// TwinCAT 3 PLC project Library
// Title: Tc3_Logging
// Company: www.peterzerlauth.com
// Author: Peter Zerlauth
// ProjectVersion: 0.0.0.0
// ProgramVersion: 3.1.4026.19
// libraries:
//   Tc2_Standard, * (Beckhoff Automation GmbH)
//   Tc2_System, * (Beckhoff Automation GmbH)
//   Tc2_Utilities, * (Beckhoff Automation GmbH)
//   Tc3_EventLogger, * (Beckhoff Automation GmbH)
//   Tc3_Module, * (Beckhoff Automation GmbH)
// project tree:
//   Helpers/ F_Format.TcPOU, F_InstancePath.TcPOU (not stored)
//   Logger/ FB_Argument.TcPOU, FB_Logger.TcPOU, I_Argument.TcIO
//   Logging/ E_LogLevel.TcDUT (not stored), FB_Logging.TcPOU, I_Logger.TcIO, I_Logging.TcIO, ST_Message.TcDUT (not stored)
//   Project Information/ F_GetCompany.TcPOU (not stored), F_GetTitle.TcPOU (not stored), F_GetVersion.TcPOU
//   TcLogging/ FB_TcLogging.TcPOU
//   Version/ Global_Version.TcGVL
// (motion and I/O tree: see PLC project plc01)
// real-time tasks:
//   TASK SlowTask: cycle T#20ms, priority 20, ADS port 350
//   TASK FastTask: cycle T#1ms, priority 1, ADS port 351

// ---- Version/Global_Version.TcGVL
{attribute 'TcGenerated'}
{attribute 'no-analysis'}
{attribute 'linkalways'}
// This function has been automatically generated from the project information.
VAR_GLOBAL CONSTANT
	{attribute 'const_non_replaced'}
	stLibVersion_Tc3_Logging : ST_LibVersion := (iMajor := 0, iMinor := 0, iBuild := 0, iRevision := 0, nFlags := 0, sVersion := '0.0.0.0');
END_VAR

// ---- Logger/I_Argument.TcIO
INTERFACE I_Argument

METHOD PUBLIC M_AddBOOL : I_Argument
VAR_INPUT
	nValue:				LINT;
END_VAR
END_METHOD

METHOD PUBLIC M_AddINT : I_Argument
VAR_INPUT
	nValue:				LINT;
END_VAR
END_METHOD

METHOD PUBLIC M_AddREAL : I_Argument
VAR_INPUT
	fValue:				LREAL;
	nDecimals:			USINT;
END_VAR
END_METHOD

METHOD PUBLIC M_AddSTRING : I_Argument
VAR_INPUT
	sValue:				STRING(255);
END_VAR
END_METHOD

METHOD PUBLIC M_AddTIME : I_Argument
VAR_INPUT
	tValue:				TIME;
END_VAR
END_METHOD

METHOD PUBLIC M_Clear : I_Argument
VAR_INPUT
END_VAR
END_METHOD

PROPERTY PUBLIC P_Value : string(255)
GET
END_GET
END_PROPERTY

END_INTERFACE

// ---- Logging/I_Logger.TcIO
INTERFACE I_Logger

METHOD PUBLIC M_AddBOOL
VAR_INPUT
	nValue:				LINT;
END_VAR
END_METHOD

METHOD PUBLIC M_AddINT
VAR_INPUT
	nValue:				LINT;
END_VAR
END_METHOD

METHOD PUBLIC M_AddREAL
VAR_INPUT
	fValue:				LREAL;
	nDecimals:			USINT;
END_VAR
END_METHOD

METHOD PUBLIC M_AddSTRING
VAR_INPUT
	sValue:				STRING(255);
END_VAR
END_METHOD

METHOD PUBLIC M_AddTIME
VAR_INPUT
	tValue:				TIME;
END_VAR
END_METHOD

METHOD PUBLIC M_Debug : BOOL
VAR_INPUT
	sMessage:			STRING(255);
END_VAR
END_METHOD

METHOD PUBLIC M_Error : BOOL
VAR_INPUT
	nID:				UDINT;
	sMessage:			STRING(255);
END_VAR
END_METHOD

METHOD PUBLIC M_Fatal : BOOL
VAR_INPUT
	nID:				UDINT;
	sMessage:			STRING(255);
END_VAR
END_METHOD

METHOD PUBLIC M_Info : BOOL
VAR_INPUT
	nID:				UDINT;
	sMessage:			STRING(255);
END_VAR
END_METHOD

METHOD PUBLIC M_Warn : BOOL
VAR_INPUT
	nID:				UDINT;
	sMessage:			STRING(255);
END_VAR
END_METHOD

END_INTERFACE

// ---- Logging/I_Logging.TcIO
INTERFACE I_Logging

METHOD PUBLIC M_Attach : BOOL
VAR_INPUT
	iLogging:				I_Logging;
END_VAR
END_METHOD

METHOD PUBLIC M_Log : BOOL
VAR_INPUT
	stMessage:			ST_Message;
END_VAR
END_METHOD

PROPERTY PUBLIC P_LogLevel : E_LogLevel
GET
END_GET
SET
END_SET
END_PROPERTY

END_INTERFACE

// ---- Helpers/F_Format.TcPOU
FUNCTION F_Format : STRING(255)
VAR_INPUT
    sMessage:				STRING(255);
    sArguments:				STRING(255);	// Arguments are separated by $R 
END_VAR
VAR
    sArg:					STRING; 	// single argument
    nPosition:				INT;         	// Position of the $R delimiter
    nPlaceholder:			INT;         	// Position of the %s placeholder
END_VAR

// replace placeholders with arguments
F_Format := sMessage;

IF sArguments = '' THEN
    RETURN;
END_IF

nPosition := FIND(sArguments, '$R');
WHILE nPosition > 0 DO
    
    sArg := LEFT(sArguments, nPosition - 1);
    
    nPlaceholder := FIND(F_Format, '%s');
    IF nPlaceholder > 0 THEN
        F_Format := REPLACE(F_Format, sArg, 2, nPlaceholder);
    ELSE
        RETURN;
    END_IF
	
    sArguments := DELETE(sArguments, nPosition, 1);
    nPosition := FIND(sArguments, '$R');
    
END_WHILE

END_FUNCTION

// ---- Logger/FB_Argument.TcPOU
FUNCTION_BLOCK FB_Argument IMPLEMENTS I_Argument
VAR_INPUT
END_VAR
VAR_OUTPUT
END_VAR
VAR
	sValue:					STRING(255); 
END_VAR

METHOD PUBLIC M_AddBOOL : I_Argument
VAR_INPUT
	nValue:				LINT;
END_VAR
sValue:= LINT_TO_STRING(nValue);			// convert
sValue:= CONCAT(sValue, '$R');				// add separator
sValue:= CONCAT(sValue, sValue);	// add new arg
M_AddBOOL:= THIS^;
END_METHOD

METHOD PUBLIC M_AddINT : I_Argument
VAR_INPUT
	nValue:				LINT;
END_VAR
VAR
	sTemp: 			STRING;
END_VAR
sTemp:= LINT_TO_STRING(nValue);			// convert
sTemp:= CONCAT(sTemp, '$R');				// add separator
sValue:= CONCAT(sValue, sTemp);	// add new arg
M_AddINT:= THIS^;
END_METHOD

METHOD PUBLIC M_AddREAL : I_Argument
VAR_INPUT
	fValue:				LREAL;
	nDecimals:			USINT;
END_VAR
VAR
	sTemp: 			STRING;
END_VAR
sTemp:= LREAL_TO_FMTSTR(fValue, nDecimals, TRUE);		// convert
sTemp:= CONCAT(sTemp, '$R');							// add separator
sValue:= CONCAT(sValue, sTemp);				// add new arg
M_AddREAL:= THIS^;
END_METHOD

METHOD PUBLIC M_AddSTRING : I_Argument
VAR_INPUT
	sValue:				STRING(255);
END_VAR
THIS^.sValue:= CONCAT(THIS^.sValue, CONCAT(sValue, '$R'));				// add separator 
M_AddSTRING:= THIS^;
END_METHOD

METHOD PUBLIC M_AddTIME : I_Argument
VAR_INPUT
	tValue:				TIME;
END_VAR
VAR
	sTemp: 			STRING;
END_VAR
sValue:= CONCAT(TIME_TO_STRING(tValue), '$R');				// add separator
sTemp:= CONCAT(sValue, sTemp);	// add new arg
M_AddTIME:= THIS^;
END_METHOD

METHOD PUBLIC M_Clear : I_Argument
VAR_INPUT
END_VAR
sValue:= '';
M_Clear:= THIS^;
END_METHOD

PROPERTY PUBLIC P_Value : string(255)
GET
P_Value:= sValue;
END_GET
END_PROPERTY

END_FUNCTION_BLOCK

// ---- Logger/FB_Logger.TcPOU
{attribute 'reflection'} 
FUNCTION_BLOCK FB_Logger
VAR_INPUT
	iLogging:			I_Logging;
END_VAR
VAR_OUTPUT
	fbArguments:				FB_Argument;
END_VAR
VAR
    {attribute 'hide'} 
    {attribute 'instance-path'} 
    {attribute 'noinit'} 
    sInstancePath:				STRING(255); 
END_VAR

//FB_Init ist immer implizit verfügbar und wird primär für die Initialisierung verwendet.
//Der Rückgabewert wird nicht ausgewertet. Für gezielte Einflussnahme können Sie
//die Methoden explizit deklarieren und darin mit dem Standard-Initialisierungscode 
//zusätzlichen Code bereitstellen. Sie können den Rückgabewert auswerten.
METHOD FB_Init: BOOL
VAR_INPUT    
bInitRetains: BOOL; // TRUE: Die Retain-Variablen werden initialisiert (Reset warm / Reset kalt)    
bInCopyCode: BOOL;  // TRUE: Die Instanz wird danach in den Kopiercode kopiert (Online-Change)
END_VAR
sInstancePath:= F_InstancePath(sInstancePath);
END_METHOD

METHOD PUBLIC M_Critical : BOOL
VAR_INPUT
	nID:				UDINT;
	sMessage:			STRING(255);
END_VAR
VAR
	stMessage:			ST_Message;
END_VAR
IF iLogging = 0 THEN
	RETURN;
END_IF

stMessage.eLogLevel:= E_LogLevel.Critical;
stMessage.nID:= nID;
stMessage.nTimestamp:= F_GetSystemTime();
stMessage.sMessage:= sMessage;
stMessage.sArguments:= fbArguments.P_Value;
stMessage.sDefault:= F_Format(sMessage, fbArguments.P_Value);
stMessage.sSource:= sInstancePath;
fbArguments.M_Clear();

iLogging.M_Log(stMessage);
END_METHOD

METHOD PUBLIC M_Error : BOOL
VAR_INPUT
	nID:				UDINT;
	sMessage:			STRING(255);
END_VAR
VAR
	stMessage:			ST_Message;
END_VAR
IF iLogging = 0 THEN
	RETURN;
END_IF

stMessage.eLogLevel:= E_LogLevel.Error;
stMessage.nID:= nID;
stMessage.nTimestamp:= F_GetSystemTime();
stMessage.sMessage:= sMessage;
stMessage.sArguments:= fbArguments.P_Value;
stMessage.sDefault:= F_Format(sMessage, fbArguments.P_Value);
stMessage.sSource:= sInstancePath;
fbArguments.M_Clear();

iLogging.M_Log(stMessage);
END_METHOD

METHOD PUBLIC M_Info : BOOL
VAR_INPUT
	nID:				UDINT;
	sMessage:			STRING(255);
END_VAR
VAR
	stMessage:			ST_Message;
END_VAR
IF iLogging = 0 THEN
	RETURN;
END_IF

stMessage.eLogLevel:= E_LogLevel.Info;
stMessage.nID:= nID;
stMessage.nTimestamp:= F_GetSystemTime();
stMessage.sMessage:= sMessage;
stMessage.sArguments:= fbArguments.P_Value;
stMessage.sDefault:= F_Format(sMessage, fbArguments.P_Value);
stMessage.sSource:= sInstancePath;
fbArguments.M_Clear();

iLogging.M_Log(stMessage);
END_METHOD

METHOD PUBLIC M_Verbose : BOOL
VAR_INPUT
	sMessage:			STRING(255);
END_VAR
VAR
	stMessage:			ST_Message;
END_VAR
IF iLogging = 0 THEN
	RETURN;
END_IF

stMessage.eLogLevel:= E_LogLevel.Verbose;
stMessage.nID:= 0;
stMessage.nTimestamp:= F_GetSystemTime();
stMessage.sMessage:= sMessage;
stMessage.sArguments:= fbArguments.P_Value;
stMessage.sDefault:= F_Format(sMessage, fbArguments.P_Value);
stMessage.sSource:= sInstancePath;
fbArguments.M_Clear();

iLogging.M_Log(stMessage);
END_METHOD

METHOD PUBLIC M_Warning : BOOL
VAR_INPUT
	nID:				UDINT;
	sMessage:			STRING(255);
END_VAR
VAR
	stMessage:			ST_Message;
END_VAR
IF iLogging = 0 THEN
	RETURN;
END_IF

stMessage.eLogLevel:= E_LogLevel.Warning;
stMessage.nID:= nID;
stMessage.nTimestamp:= F_GetSystemTime();
stMessage.sMessage:= sMessage;
stMessage.sArguments:= fbArguments.P_Value;
stMessage.sDefault:= F_Format(sMessage, fbArguments.P_Value);
stMessage.sSource:= sInstancePath;
fbArguments.M_Clear();

iLogging.M_Log(stMessage);
END_METHOD

PROPERTY PUBLIC P_Argument : I_Argument
GET
P_Argument:= fbArguments;
END_GET
END_PROPERTY

PROPERTY PUBLIC P_Logger : I_Logging
GET
P_Logger:= iLogging;
END_GET
SET
iLogging:= P_Logger;
END_SET
END_PROPERTY

END_FUNCTION_BLOCK

// ---- Logging/FB_Logging.TcPOU
// Provide logging 
FUNCTION_BLOCK FB_Logging IMPLEMENTS I_Logging
VAR_INPUT
	eLogLevel:				E_LogLevel:= E_LogLevel.Verbose;
END_VAR
VAR_OUTPUT
    bInfo:					BOOL;
    bWarning:				BOOL;
    bError:					BOOL;
    bCritical:				BOOL;
END_VAR
VAR
	aMessages:				ARRAY[0..99] OF ST_Message; // Message store
    nMessages:				UINT := 0;                     // Message count
	{attribute 'hide'} 
	nIndex: 				UINT;
	iLogging:				I_Logging;
END_VAR

nIndex := 0;
WHILE nIndex < nMessages DO
	IF aMessages[nIndex].bActive THEN
		aMessages[nIndex].bActive:= FALSE;
		nIndex := nIndex + 1;
	ELSE
		IF iLogging <> 0 THEN
			// publish outdated messages to remove
			iLogging.M_Log(aMessages[nIndex]);
		END_IF
        MEMMOVE(ADR(aMessages[nIndex]), ADR(aMessages[nIndex + 1]), SIZEOF(ST_Message) * (nMessages - nIndex));
        nMessages := nMessages - 1;
		bInfo:=	FALSE;
		bWarning:=	FALSE;
		bError:= FALSE;
		bCritical:= FALSE;
    END_IF
END_WHILE

METHOD PUBLIC M_Attach : BOOL
VAR_INPUT
	iLogging:				I_Logging;
END_VAR
IF THIS^.iLogging = 0 THEN
	THIS^.iLogging:= iLogging;
	M_Attach:= TRUE;
ELSIF THIS^.iLogging = iLogging THEN
	// already inside
	M_Attach:= TRUE;
	RETURN;
ELSE
	// redirect to next logging function block
	THIS^.iLogging.M_Attach(iLogging);
END_IF
END_METHOD

METHOD PUBLIC M_Log : BOOL
VAR_INPUT
	stMessage:			ST_Message;
END_VAR
VAR
END_VAR
IF eLogLevel > stMessage.eLogLevel THEN
	M_Log:= TRUE;
	RETURN;
END_IF

CASE stMessage.eLogLevel OF
	E_LogLevel.Info:
    	bInfo:= TRUE;
		
	E_LogLevel.Warning:		
    	bWarning:= TRUE;
		
	E_LogLevel.Error:
    	bError:= TRUE;
		
	E_LogLevel.Critical:
    	bCritical:= TRUE;
		
	ELSE
		;
END_CASE


// Find
FOR nIndex := 0 TO nMessages DO
    IF aMessages[nIndex].sMessage = stMessage.sMessage AND_THEN aMessages[nIndex].sSource = stMessage.sSource THEN
        aMessages[nIndex].bActive:= TRUE;
		M_Log := TRUE;
        RETURN;
    END_IF
END_FOR

// else Add
IF nMessages < 99 THEN
	nIndex := nMessages;
	stMessage.bActive:= TRUE;
    aMessages[nMessages]:= stMessage;;
    nMessages := nMessages + 1;
	// reduce internal buffers 
	// publish new messages to log
	IF iLogging <> 0 THEN
		iLogging.M_Log(stMessage);
	END_IF
	M_Log := TRUE;
END_IF
END_METHOD

PROPERTY PUBLIC P_LogLevel : E_LogLevel
GET
P_LogLevel:= eLogLevel;
END_GET
SET
eLogLevel:= P_LogLevel;
END_SET
END_PROPERTY

END_FUNCTION_BLOCK

// ---- Project Information/F_GetVersion.TcPOU
// This function has been automatically generated from the project information.
{attribute 'signature_flag' := '1073741824'}
{attribute 'TcGenerated'}
{attribute 'no-analysis'}
FUNCTION F_GetVersion : ST_LibVersion
VAR_INPUT
	
END_VAR

F_GetVersion.iMajor := 0;
F_GetVersion.iMinor := 0;
F_GetVersion.iBuild := 0;
F_GetVersion.iRevision := 0;
F_GetVersion.sVersion := '0.0.0.0';
F_GetVersion.nFlags := 0;

END_FUNCTION

// ---- TcLogging/FB_TcLogging.TcPOU
// Provide logging 
FUNCTION_BLOCK FB_TcLogging IMPLEMENTS I_Logging
VAR_INPUT
	eLogLevel:				E_LogLevel:= E_LogLevel.Verbose;
END_VAR
VAR_OUTPUT
END_VAR
VAR
	iLogging:				I_Logging;
END_VAR

METHOD PUBLIC M_Attach : BOOL
VAR_INPUT
	iLogging:				I_Logging;
END_VAR
IF THIS^.iLogging = 0 THEN
	THIS^.iLogging:= iLogging;
	M_Attach:= TRUE;
ELSIF THIS^.iLogging = iLogging THEN
	// already inside
	M_Attach:= TRUE;
	RETURN;
ELSE
	// redirect to next logging function block
	THIS^.iLogging.M_Attach(iLogging);
END_IF
END_METHOD

METHOD PUBLIC M_Log : BOOL
VAR_INPUT
	stMessage:			ST_Message;
END_VAR
VAR
	fbMsg:				FB_TcMessage; 
	fbSourceInfo:		FB_TcSourceInfo;
END_VAR
IF THIS^.eLogLevel > eLogLevel THEN
	M_Log:= TRUE;
	RETURN;
END_IF

IF stMessage.bActive THEN

	fbSourceInfo.Clear();
	fbSourceInfo.sName:= stMessage.sSource;
	
	CASE stMessage.eLogLevel OF
		E_LogLevel.Verbose:
			fbMsg.CreateEx(TC_EVENTS.TcLogging.Verbose, fbSourceInfo); 	
	
		E_LogLevel.Info:
			fbMsg.CreateEx(TC_EVENTS.TcLogging.Info, fbSourceInfo); 
			
		E_LogLevel.Warning:		
			fbMsg.CreateEx(TC_EVENTS.TcLogging.Warning, fbSourceInfo); 
			
		E_LogLevel.Error:
			fbMsg.CreateEx(TC_EVENTS.TcLogging.Error, fbSourceInfo); 
			
		E_LogLevel.Critical:
			fbMsg.CreateEx(TC_EVENTS.TcLogging.Critical, fbSourceInfo); 
			
	END_CASE
	
	fbMsg.ipArguments.Clear().AddString(stMessage.sDefault);
	
	fbMsg.Send(stMessage.nTimestamp);

END_IF
END_METHOD

PROPERTY PUBLIC P_LogLevel : E_LogLevel
GET
P_LogLevel:= eLogLevel;
END_GET
SET
eLogLevel:= P_LogLevel;
END_SET
END_PROPERTY

END_FUNCTION_BLOCK
